TYPE ST_TrafficLightInput :
STRUCT

	bDayMode : BOOL;
	bSetRed : BOOL;
	bSetGreen : BOOL;
END_STRUCT
END_TYPE

(* stored: Version 1.1.0.1, ProductVersion 3.1.4024.0
   DUT ST_TrafficLightInput: Id {e56f1dc8-4a56-4c98-a9aa-3554ae6cdab8} *)
